SUBAPPLICATION Uebung_015_AX (* Object Pointer umschalten *)
  (* Standard: 61499-2; Description: Copyright (c) 2026 Meisterschulen am Ostbahnhof This program and the accompanying materials are made available under the terms of the Eclipse Public License 2.0 which is available at https://www.eclipse.org/legal/epl-2.0/ SPDX-License-Identifier: EPL-2.0 *)
  (* Version 1.0, 2026-09-10, Franz Höpfinger, Meisterschulen am Ostbahnhof, initial API and implementation and/or initial documentation *)
  PACKAGE Uebungen;
  IMPORT isobus::UT::io::Softkey::SoftKeyActivationCode::SK_RELEASED;
  IMPORT Uebungen::const::UT::DefaultPool::Button_A1;
  IMPORT Uebungen::const::UT::DefaultPool::ObjectPointer_P1;
  IMPORT Uebungen::const::UT::DefaultPool::SoftKey_F1;
  IMPORT Uebungen::const::UT::DefaultPool::SoftKey_F2;
  IMPORT isobus::UT::Q::const::IDs::ID_NULL;
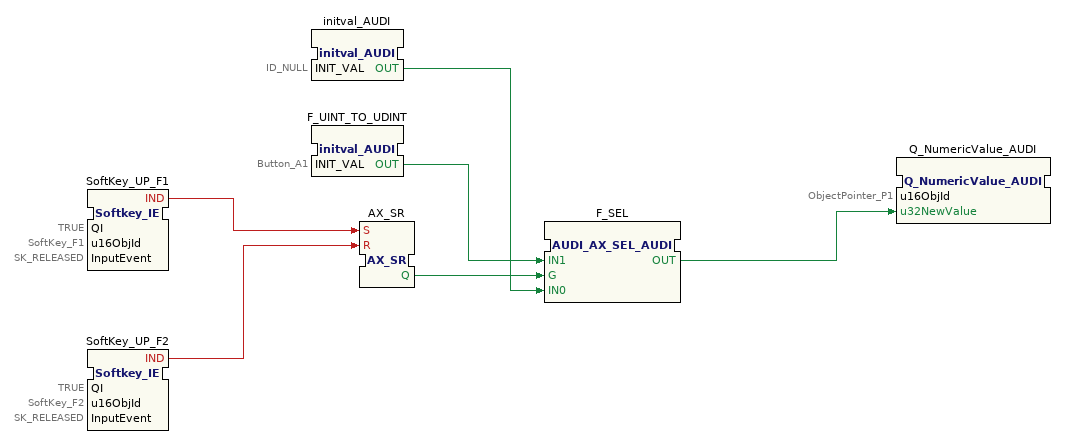
  FBS
    SoftKey_UP_F1 : isobus::UT::io::Softkey::Softkey_IE(QI := TRUE, u16ObjId := SoftKey_F1, InputEvent := SK_RELEASED);
    SoftKey_UP_F2 : isobus::UT::io::Softkey::Softkey_IE(QI := TRUE, u16ObjId := SoftKey_F2, InputEvent := SK_RELEASED);
    AX_SR : adapter::events::unidirectional::AX_SR;
    F_UINT_TO_UDINT : adapter::types::unidirectional::AUDI::initval::initval_AUDI(INIT_VAL := Button_A1);
    F_SEL : adapter::iec61131::selection::AUDI_AX_SEL_AUDI;
    Q_NumericValue_AUDI : isobus::UT::Q::Q_NumericValue_AUDI(u16ObjId := ObjectPointer_P1);
    initval_AUDI : adapter::types::unidirectional::AUDI::initval::initval_AUDI(INIT_VAL := ID_NULL);
  END_FBS
  EVENT_CONNECTIONS
    SoftKey_UP_F1.IND TO AX_SR.S;
    SoftKey_UP_F2.IND TO AX_SR.R;
  END_CONNECTIONS
  ADAPTER_CONNECTIONS
    F_UINT_TO_UDINT.OUT TO F_SEL.IN1;
    AX_SR.Q TO F_SEL.G;
    initval_AUDI.OUT TO F_SEL.IN0;
    F_SEL.OUT TO Q_NumericValue_AUDI.u32NewValue;
  END_CONNECTIONS
END_SUBAPPLICATION
